PROGRAM P0_00_MAIN
VAR
	test1: BOOL;
	test2: BOOL;
	test3: BOOL;
	test: BOOl;
END_VAR

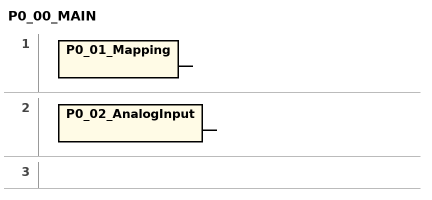
// NETWORK 1
P0_01_Mapping();

// NETWORK 2
P0_02_AnalogInput();

// NETWORK 3

END_PROGRAM

(* stored: Version 1.1.0.1, ProductVersion 3.1.4024.12
   POU P0_00_MAIN: Id {86ce4e51-607a-4571-99ad-8e912cffc189}, SpecialFunc None *)
